PROGRAM MAIN
VAR
	MySystem : FB_Systems;
END_VAR

MySystem();

END_PROGRAM

(* stored: Version 1.1.0.1, ProductVersion 3.1.4024.16
   POU MAIN: Id {92f14351-dcbb-423d-9f1d-1757ec898e20}, SpecialFunc None
   Folder VISUs: Id {a11fb6ec-be5a-0119-390f-50fc7439d0c0} *)
